//---------------------------------------------------------------------------------------------------------------
//
//  HAUD 2024.11.21
//
//
//  fb_Instance
//-----------------------------------------------------------------------------
//  - base class for my process instance to work with fb_ProcessCollector
//
//  - _nProcess --> whoami, this is me
//
//  - fb_ProcessCollector[_nProcess].Cycle() is called in APPLICATION(PRG)
//    - handles range of XtsStations
//    - range must be closed and in consecutive order
//
//    - combines states into bitmasks, one bit per XtsStation
//    - controls forwarding of commands to range of XtsStations 
//      (see fb_ProcessCollector.Cycle())
//
//  - reference to all _ItfProcessCollector(I_ProcessCollector)[]
//    - _ItfProcessCollector[nProcess] Get/Set properties and methods
//
//  - Control / State of my process
//    - datafield for control and state provided
//    - _Ctrl 
//      --> commands to my process; fb_ProcessCollector[_nProcess]
//      --> is linked (REF=) automatically in Check()
//
//      Cmd               : E_PROCESS_CTRL; // command enum for my process
//      ProcessTarget     : UINT;           // target of my process
//      ActivateStation   : WORD;           // is checked for every job
//                                          // every bit is a XtsStation
//
//      NestMask          : BYTE;           // one mask for all XtsStations
//      - every bit is a PosStop in a XtsStation
//      - copied to every XtsStation in my process when movers are about to leave
//
//    - _State
//      --> satus information from my process
//      --> check for plausible StationLast / StationFirst range of XtsStations
//
//      State             : E_PROCESS_STATE;  // state enuum from my process
//      Result            : E_PROGRESS;       // substate from my process, BUSY signals state is ready for interaction
//      Check             : E_PROCESS_CHECK;  // plausibility check of StationLast and StationFirst 
//
//
//  - basic check and var names, so you can build your procedures with it
//
//  - processes may be connected via linked list, you decide.
//    - linked list for processes is intended to work as job buffer
//    - linked list provides information via ST_PROCESS_DATA, 
//      add what you have to in there
//    - linked ist to all process instances provided
//
//  - inherit this base class for your application, call Check() cyclic
//
//---------------------------------------------------------------------------------------------------------------//
// This SOFTWARE is provided as an Exemple by THE PROVIDER "as is" and "with all faults." THE PROVIDER makes no  //
// representations or warranties of any kind concerning the safety, suitability, lack of viruses, inaccuracies,  //
// typographical errors, or other harmful components of this SOFTWARE. There are inherent dangers in the use of  //
// any software, and you are solely responsible for determining whether this SOFTWARE is compatible with your    //
// equipment and other software installed on your equipment. You are also solely responsible for the protection  //
// of your equipment and backup of your data, and THE PROVIDER will not be liable for any damages you may suffer //
// in connection with using, modifying, or distributing this SOFTWARE.                                           //
//---------------------------------------------------------------------------------------------------------------//
FUNCTION_BLOCK fb_Instance
VAR
  // process index
  _nProcess               : E_INSTANCE;           // whoami

  _InstanceCtrl           : REFERENCE TO ARRAY[1..MAX_PROCESS] OF ST_INSTANCE_CTRL;
  _InstanceState          : REFERENCE TO ARRAY[1..MAX_PROCESS] OF ST_INSTANCE_STATE;

  _eCmd,
  _eCmdOld                : E_INSTANCE_CMD;       // commands for local state machine
  _eStateInstance         : E_INSTANCE_STATE;     // local state machine for infeed procedure

  _eResult,
  _eStateProgress         : E_PROGRESS;           // substate for lacal state machine

  _eInit                  : E_PROGRESS;           // startup
  _eCheck                 : E_INSTANCE_CHECK;     // pointer checks


  // local ctrl / state datafields for you to use, connected by reference to _ItfProcessCollector[_nProcess]
  _Ctrl                   : ST_PROCESS_CTRL;      // control to write, connected by reference to _ItfProcessCollector
  _State                  : ST_PROCESS_STATE;     // state   to read,  connected by reference to _ItfProcessCollector

  _ItfProcessCollector    : ARRAY[1..MAX_PROCESS] OF I_ProcessCollector;    // information and configuration of the connected ProcessCollector for given range of XtsStations

  _ItfProcessList         : ARRAY[1..MAX_PROCESS] OF I_Process_LinkedList;  // access to all linked lists for process entry
  _ListResult             : ST_PROCESS_LIST_RESULT;
  _ProcessData            : ST_PROCESS_DATA;

  {attribute 'displaymode':='bin'}
  _wTargetMask            : ARRAY[1..SIZEOF(T_PROCESS)*8] OF BYTE; // bits for PosStop[] to use in XtsStation of target process

  _stMsg                  : ST_Message;
  _MessageLevel           : E_MessageType;
END_VAR

METHOD Check : BOOL // call this method in the extending/inheriting class
//-----------------------------------------------------------------------------
//-----------------------------------------------------------------------------
// plausibility checks
//-----------------------------------------------------------------------------
IF NOT (_nProcess > 0)
THEN
  _eCheck                 := E_INSTANCE_CHECK.INVALID_PROCESS_ID_ZERO;
  RETURN;
END_IF

IF NOT (_nProcess < E_INSTANCE.INSTANCE_MAX)
THEN
  _eCheck                 := E_INSTANCE_CHECK.INVALID_PROCESS_ID_MAX;
  RETURN;
END_IF
//-----------------------------------------------------------------------------
//-----------------------------------------------------------------------------
// pointer checks
//-----------------------------------------------------------------------------
IF NOT __ISVALIDREF(_InstanceCtrl)
THEN
  _eCheck                 := E_INSTANCE_CHECK.INVALID_INSTANCE_CONTROL_REFERENCE;
  RETURN;
END_IF

IF NOT __ISVALIDREF(_InstanceState)
THEN
  _eCheck                 := E_INSTANCE_CHECK.INVALID_INSTANCE_STATE_REFERENCE;
  RETURN;
END_IF

IF NOT (_ItfProcessCollector[_nProcess] <> 0) 
THEN
  _eCheck                 := E_INSTANCE_CHECK.INVALID_INTERFACE_POINTER;
  RETURN;
END_IF

IF NOT (_ItfProcessCollector[_nProcess].ProcessId > 0)
THEN
  _eCheck                 := E_INSTANCE_CHECK.INVALID_PROCESS_ID_ZERO;
  RETURN;
END_IF

IF NOT (_ItfProcessCollector[_nProcess].ProcessId < E_INSTANCE.INSTANCE_MAX)
THEN
  _eCheck                 := E_INSTANCE_CHECK.INVALID_PROCESS_ID_MAX;
  RETURN;
END_IF

IF NOT (_nProcess = _ItfProcessCollector[_nProcess].ProcessId)
THEN
  _eCheck                 := E_INSTANCE_CHECK.INVALID_PROCESS_ID_NOTEQUAL_COLLECTOR_ID;
  RETURN;
END_IF

IF NOT (_ItfProcessList[_nProcess] <> 0)
THEN
  _eCheck                 := E_INSTANCE_CHECK.INVALID_INDEX_IN_LIST;
  RETURN;
END_IF
//-----------------------------------------------------------------------------
//-----------------------------------------------------------------------------
// connect datafields to interface of ProcessCollector
//-----------------------------------------------------------------------------
_ItfProcessCollector[_nProcess].ProcessCtrl   REF= _Ctrl;
_ItfProcessCollector[_nProcess].ProcessState  REF= _State;

//-----------------------------------------------------------------------------
//-----------------------------------------------------------------------------
// set message device
//-----------------------------------------------------------------------------
_stMsg.eDevice            := e_Device.Process + TO_UINT(_nProcess);
//-----------------------------------------------------------------------------
//-----------------------------------------------------------------------------
_eCheck                   := E_INSTANCE_CHECK.CHECK_DONE;
Check                     := TRUE;
END_METHOD

PROPERTY CollectorInterface : array[1..MAX_PROCESS] of I_ProcessCollector
SET
_ItfProcessCollector := CollectorInterface;
END_SET
END_PROPERTY

PROPERTY InstanceCtrl : REFERENCE TO ARRAY[1..MAX_PROCESS] OF ST_INSTANCE_CTRL
SET
_InstanceCtrl ref= InstanceCtrl;
END_SET
END_PROPERTY

PROPERTY InstanceState : REFERENCE TO ARRAY[1..MAX_PROCESS] OF ST_INSTANCE_STATE
SET
_InstanceState ref= InstanceState;
END_SET
END_PROPERTY

PROPERTY ProcessId : E_INSTANCE
GET
ProcessId := _nProcess;
END_GET
SET
_nProcess := ProcessId;
END_SET
END_PROPERTY

PROPERTY ProcessLinkedLists : ARRAY[1..max_process] OF I_Process_LinkedList
SET
_ItfProcessList := ProcessLinkedLists;
END_SET
END_PROPERTY

END_FUNCTION_BLOCK

(* stored: Version 1.1.0.1, ProductVersion 3.1.4024.15
   POU fb_Instance: Id {02367fcb-67b8-497b-8382-1c3639f01a80}, SpecialFunc None
   Folder properties: Id {5f969983-7274-474e-ad53-ecf15d94990d}
   Method Check: Id {04192027-e492-4023-92ca-671af767f088}
   Property CollectorInterface: Id {7856fb23-1ef1-472e-9855-7bec6a7c2039}
   Set Set: Id {d83e93f2-0907-4e4e-899d-c33bd6f05c59}
   Property InstanceCtrl: Id {db5cb503-c126-4bf4-9d9e-33d5513507b6}
   Set Set: Id {eaba3005-7366-4abe-8b29-c097c6288b47}
   Property InstanceState: Id {24069783-085b-4d3c-814f-09ba43146601}
   Set Set: Id {dea38988-006a-4feb-a9dc-eb0cdbca8050}
   Property ProcessId: Id {bc02b386-af4a-427a-bfae-f03f977e543e}
   Get Get: Id {f26a4457-27eb-4b2a-bb3e-26741e3e8a80}
   Set Set: Id {82f5dac8-30d1-408a-8463-5b7d3dbc951d}
   Property ProcessLinkedLists: Id {f1f4c45b-0247-4e47-9cfc-0c8d3318a647}
   Set Set: Id {d5137f63-8b56-4b2c-a086-29d9076bed68} *)
